TYPE U_Convert_UDINT32 :
UNION
	nValue		:UDINT;
	arrByte		:ARRAY[1..4] OF BYTE;
END_UNION
END_TYPE

(* stored: Version 1.1.0.1, ProductVersion 3.1.4024.12
   DUT U_Convert_UDINT32: Id {ef136247-0211-4106-92f2-2d517c91549e} *)
